// TIA Portal project "Test2" (V18)

(* hardware
DEVICE "PC-System_1"  SIMATIC PC station
   slot 0: "SIMATIC PC station"  Rail  SIMATIC PC-Station  V1.0
      slot 125: "Stationmanager"  Station_Manager  V6.0.4
   slot 1: "HMI_RT_1"  WinCC RT Professional  6AV2 105-0xxxx-xxxx  18.0.0.0
   slot 2: "IE general_1"  IE General  IE_CP  V8.2.0
      slot 1: "PROFINET interface"  IEGeneral.Interface.8.2.0
DEVICE "S7-1500/ET200MP station_1"  S7-1500 station
   slot 0: "Rail_0"  Rack  6ES7 590-1***0-0AA0
   slot 1: "PLC_2"  CPU 1511C-1 PN  6ES7 511-1CK01-0AB0  V2.9
      slot 3: "CPU display_1"  6ES7591-1AA00-0AA0
      slot 32768: "PROFINET interface_1"  X1
         slot 32769: "Port_1"  X1 P1
         slot 32770: "Port_2"  X1 P2
      slot 34817: "Virtual CP interface port_1"  Virtual CP interface port  Virtual CP interface port
*)

// ===== PLC "PLC_2"  CPU 1511C-1 PN =====

VAR_GLOBAL   // PLC tag table "Default tag table"
   "L" AT %IW2 : Int;   // уровень
   "LOV-1" AT %Q4.0 : Bool;   // КЛАПАН НА ЗАКАЧКУ ВОДЫ
   "LOV-2" AT %Q4.1 : Bool;   // Клапан на выкачку
   "tag_SpeadLminus_cm_s" AT %MD1 : Real;
   "tag_SpeadLminus_cm_s_X" AT %MD2 : Real;
   "tag_SpeadLplus_cm_s" AT %MD6 : Real;
   "tag_T1_Q" AT %M17.1 : Bool;
   "tag_T1_Start" AT %M17.0 : Bool;
END_VAR

VAR_GLOBAL   // PLC tag table "E333"
   "Auto_man_LOV-1" AT %M0.1 : Bool;   // В автоманте - 1. В ручном - 0
   "Start_stop" AT %M0.2 : Bool;   // пуск-остановка клапана закачки
   "Start_stop_2" AT %M0.3 : Bool;   // Ручное упарвеление Клапаном
   "Start_stop_Nasos" AT %M0.4 : Bool;
   "Nasos(1)" AT %M0.5 : Bool;
   "Auto_man_LOV-2" AT %M0.6 : Bool;
   "Auto_man_NASOS-1" AT %M0.7 : Bool;
   "Auto_man_ALL" AT %M10.0 : Bool;
END_VAR

DATA_BLOCK "DB_1"   // DB2
{ S7_Optimized_Access := 'FALSE' }
VERSION : 0.1
   VAR
      ResetPID : Bool;
      ManOn : Bool;
      Circle_2 : Time := T#1s;
      Circle_1 : Time := T#1s;
      Level_Sim : Real;
      SetPoin_1 : Real := 0.0;
      Gain_1 : Real := -2.0;
      Gain_2 : Real := -2.0;
      TI_1 : Time := T#20ms;
      TI_2 : Time := T#20ms;
      PID_OUT_1 : Real;
      PID_OUT_2 : Real;
      Level_Sim_Dint : DInt;
      Deadband_1 : Real;
      Deadband_2 : Real;
      PID_OUT_1_dev10 : Real;
      SpeadPLUS : Real := 1.0;
      SpeadLminus : Real := 5.0;
      PID_OUT_1_Dint : DInt;
   END_VAR
BEGIN
END_DATA_BLOCK

DATA_BLOCK "Data_E333"   // DB3
{ S7_Optimized_Access := 'TRUE' }
VERSION : 0.1
   VAR
      MAX_lvl : Real := 100.0;
      MIN_lvl : Real := 0.0;
      Pump_POWER : Real;
      MAX_Uroven : Real;
      MIN_Uroven : Real;
   END_VAR
BEGIN
END_DATA_BLOCK

DATA_BLOCK "NASOS_BD"   // DB4
{ S7_Optimized_Access := 'TRUE' }
VERSION : 0.1
   VAR
      Speed_NOW : Real;
   END_VAR
BEGIN
END_DATA_BLOCK

DATA_BLOCK "LOVs_DB"   // DB5
{ S7_Optimized_Access := 'TRUE' }
VERSION : 0.1
BEGIN
END_DATA_BLOCK

DATA_BLOCK "Avtonomiya_1"   // DB6
{ S7_Optimized_Access := 'TRUE' }
VERSION : 0.1
   VAR
      ZakachkaFlow : Real;
      OtkachkaFlow : Real;
   END_VAR
BEGIN
END_DATA_BLOCK

FUNCTION "LOV_1" : Void   // FC1, LAD
{ S7_Optimized_Access := 'TRUE' }
VERSION : 0.1
   VAR_TEMP
      "#DrainFlow_1" : Bool;
   END_VAR
BEGIN

REGION Network 1: КЛАПАН НА ЗАКАЧКУ ВОДЫ
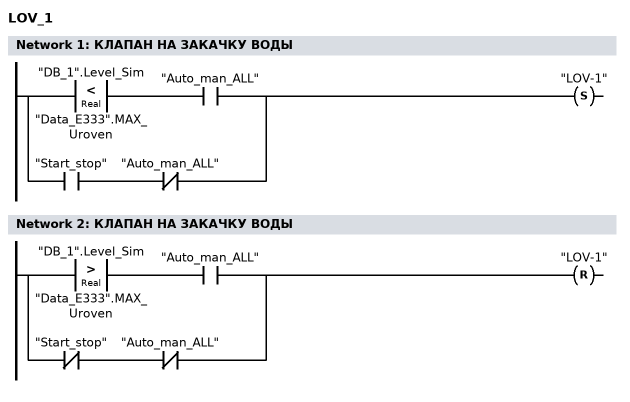
   RUNG wire#powerrail
      { S7_Templates := "SrcType := Real" } LT_Contact(in1 := "DB_1".Level_Sim, in2 := "Data_E333".MAX_Uroven)
      Contact( "Auto_man_ALL" )
      wire#w1
      S_Coil( "LOV-1" )
   END_RUNG
   RUNG wire#powerrail
      Contact( "Start_stop" )
      I_Contact( "Auto_man_ALL" )
   END_RUNG wire#w1
   // the same network as SCL:
   IF (("DB_1".Level_Sim < "Data_E333".MAX_Uroven) AND "Auto_man_ALL") OR ("Start_stop" AND NOT "Auto_man_ALL") THEN
       "LOV-1" := TRUE;
   END_IF;
END_REGION

REGION Network 2: КЛАПАН НА ЗАКАЧКУ ВОДЫ
   RUNG wire#powerrail
      { S7_Templates := "SrcType := Real" } GT_Contact(in1 := "DB_1".Level_Sim, in2 := "Data_E333".MAX_Uroven)
      Contact( "Auto_man_ALL" )
      wire#w1
      R_Coil( "LOV-1" )
   END_RUNG
   RUNG wire#powerrail
      I_Contact( "Start_stop" )
      I_Contact( "Auto_man_ALL" )
   END_RUNG wire#w1
   // the same network as SCL:
   IF (("DB_1".Level_Sim > "Data_E333".MAX_Uroven) AND "Auto_man_ALL") OR (NOT "Start_stop" AND NOT "Auto_man_ALL") THEN
       "LOV-1" := FALSE;
   END_IF;
END_REGION
END_FUNCTION

FUNCTION "FC_PID" : Void   // FC2, LAD
{ S7_Optimized_Access := 'TRUE' }
VERSION : 0.1
BEGIN

REGION Network 1
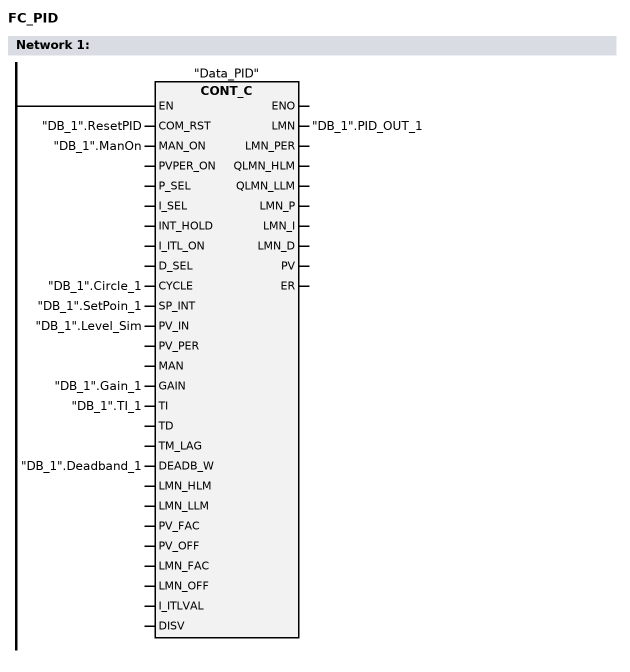
   "Data_PID"(COM_RST := "DB_1".ResetPID,   // CONT_C
              MAN_ON := "DB_1".ManOn,
              CYCLE := "DB_1".Circle_1,
              SP_INT := "DB_1".SetPoin_1,
              PV_IN := "DB_1".Level_Sim,
              GAIN := "DB_1".Gain_1,
              TI := "DB_1".TI_1,
              DEADB_W := "DB_1".Deadband_1,
              LMN => "DB_1".PID_OUT_1);
END_REGION
END_FUNCTION

FUNCTION "NASOS" : Void   // FC3, LAD
{ S7_Optimized_Access := 'TRUE' }
VERSION : 0.1
   VAR_TEMP
      PumpPower : Real;
      DrainFlow_1 : Real;
      DeltaLevel : Real;
   END_VAR
BEGIN

REGION Network 1
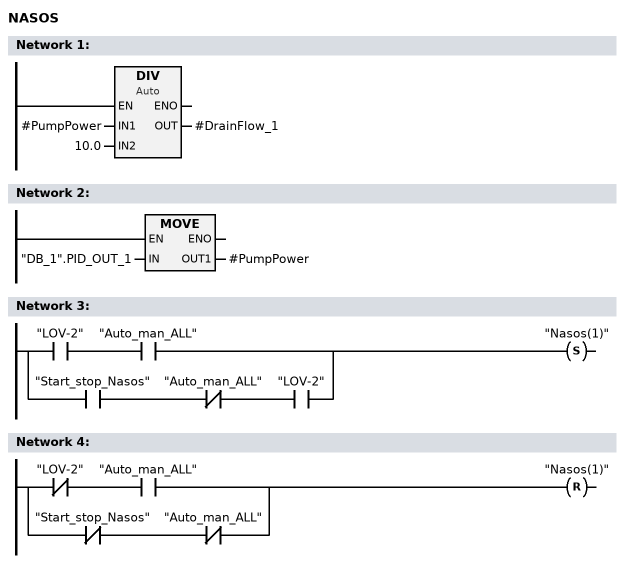
   RUNG wire#powerrail
      Div(in1 := #PumpPower, in2 := 10.0, out => #DrainFlow_1)
   END_RUNG
   // the same network as SCL:
   #DrainFlow_1 := #PumpPower / 10.0;
END_REGION

REGION Network 2
   RUNG wire#powerrail
      Move(in := "DB_1".PID_OUT_1, out1 => #PumpPower)
   END_RUNG
   // the same network as SCL:
   #PumpPower := "DB_1".PID_OUT_1;
END_REGION

REGION Network 3
   RUNG wire#powerrail
      Contact( "LOV-2" )
      Contact( "Auto_man_ALL" )
      wire#w1
      S_Coil( "Nasos(1)" )
   END_RUNG
   RUNG wire#powerrail
      Contact( "Start_stop_Nasos" )
      I_Contact( "Auto_man_ALL" )
      Contact( "LOV-2" )
   END_RUNG wire#w1
   // the same network as SCL:
   IF ("LOV-2" AND "Auto_man_ALL") OR ("Start_stop_Nasos" AND NOT "Auto_man_ALL" AND "LOV-2") THEN
       "Nasos(1)" := TRUE;
   END_IF;
END_REGION

REGION Network 4
   RUNG wire#powerrail
      I_Contact( "LOV-2" )
      Contact( "Auto_man_ALL" )
      wire#w1
      R_Coil( "Nasos(1)" )
   END_RUNG
   RUNG wire#powerrail
      I_Contact( "Start_stop_Nasos" )
      I_Contact( "Auto_man_ALL" )
   END_RUNG wire#w1
   // the same network as SCL:
   IF (NOT "LOV-2" AND "Auto_man_ALL") OR (NOT "Start_stop_Nasos" AND NOT "Auto_man_ALL") THEN
       "Nasos(1)" := FALSE;
   END_IF;
END_REGION

REGION Network 5 (SCL)
   "DB_1".Level_Sim := "DB_1".Level_Sim + ("Avtonomiya_1".ZakachkaFlow / 60.0) * 0.1
   - ("Avtonomiya_1".OtkachkaFlow  / 60.0) * ("DB_1".PID_OUT_1 / 100.0) * 0.1;

   "NASOS_BD".Speed_NOW := "Avtonomiya_1".OtkachkaFlow * ("DB_1".PID_OUT_1 / 100.0);


   "Data_E333".Pump_POWER := #PumpPower;
END_REGION
END_FUNCTION

FUNCTION "LOV_2" : Void   // FC4, LAD
{ S7_Optimized_Access := 'TRUE' }
VERSION : 0.1
BEGIN

REGION Network 1: Клапан на выкачку
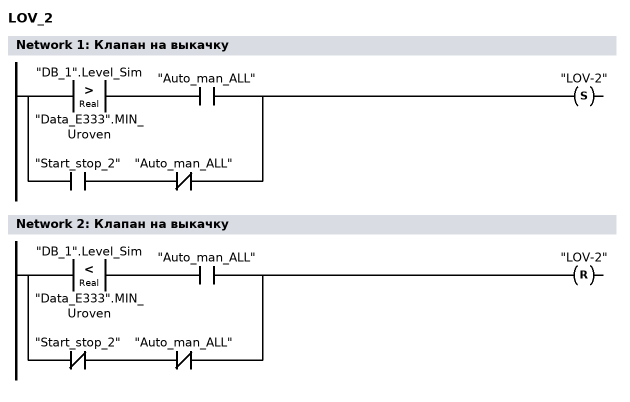
   RUNG wire#powerrail
      { S7_Templates := "SrcType := Real" } GT_Contact(in1 := "DB_1".Level_Sim, in2 := "Data_E333".MIN_Uroven)
      Contact( "Auto_man_ALL" )
      wire#w1
      S_Coil( "LOV-2" )
   END_RUNG
   RUNG wire#powerrail
      Contact( "Start_stop_2" )
      I_Contact( "Auto_man_ALL" )
   END_RUNG wire#w1
   // the same network as SCL:
   IF (("DB_1".Level_Sim > "Data_E333".MIN_Uroven) AND "Auto_man_ALL") OR ("Start_stop_2" AND NOT "Auto_man_ALL") THEN
       "LOV-2" := TRUE;
   END_IF;
END_REGION

REGION Network 2: Клапан на выкачку
   RUNG wire#powerrail
      { S7_Templates := "SrcType := Real" } LT_Contact(in1 := "DB_1".Level_Sim, in2 := "Data_E333".MIN_Uroven)
      Contact( "Auto_man_ALL" )
      wire#w1
      R_Coil( "LOV-2" )
   END_RUNG
   RUNG wire#powerrail
      I_Contact( "Start_stop_2" )
      I_Contact( "Auto_man_ALL" )
   END_RUNG wire#w1
   // the same network as SCL:
   IF (("DB_1".Level_Sim < "Data_E333".MIN_Uroven) AND "Auto_man_ALL") OR (NOT "Start_stop_2" AND NOT "Auto_man_ALL") THEN
       "LOV-2" := FALSE;
   END_IF;
END_REGION
END_FUNCTION

FUNCTION "Avtonomiya" : Void   // FC5, LAD
{ S7_Optimized_Access := 'TRUE' }
VERSION : 0.1
BEGIN

REGION Network 1
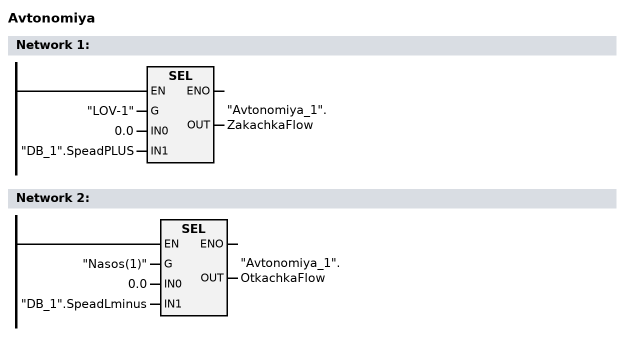
   "Avtonomiya_1".ZakachkaFlow := SEL(G := "LOV-1", IN0 := 0.0, IN1 := "DB_1".SpeadPLUS);
END_REGION

REGION Network 2
   "Avtonomiya_1".OtkachkaFlow := SEL(G := "Nasos(1)", IN0 := 0.0, IN1 := "DB_1".SpeadLminus);
END_REGION
END_FUNCTION

ORGANIZATION_BLOCK "Main"   // OB1, LAD, ProgramCycle
TITLE = "Main Program Sweep (Cycle)"
{ S7_Optimized_Access := 'TRUE' }
VERSION : 0.1
   VAR_INPUT
      Initial_Call : Bool;   // Initial call of this OB
      Remanence : Bool;   // =True, if remanent data are available
   END_VAR
   VAR_TEMP
      Temp : Real;
   END_VAR
BEGIN
END_ORGANIZATION_BLOCK

ORGANIZATION_BLOCK "PID_1"   // OB123, LAD, ProgramCycle
TITLE = "Main Program Sweep (Cycle)"
{ S7_Optimized_Access := 'TRUE' }
VERSION : 0.1
   VAR_INPUT
      Initial_Call : Bool;   // Initial call of this OB
      Remanence : Bool;   // =True, if remanent data are available
   END_VAR
BEGIN

REGION Network 1
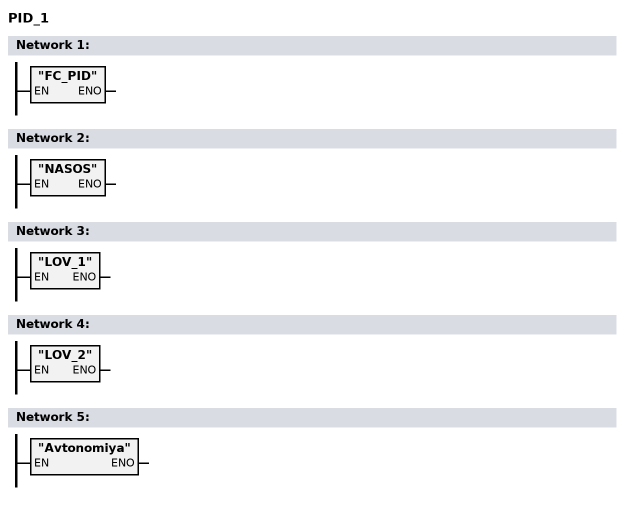
   RUNG wire#powerrail
      "FC_PID"()
   END_RUNG
   // the same network as SCL:
   "FC_PID"();
END_REGION

REGION Network 2
   RUNG wire#powerrail
      "NASOS"()
   END_RUNG
   // the same network as SCL:
   "NASOS"();
END_REGION

REGION Network 3
   RUNG wire#powerrail
      "LOV_1"()
   END_RUNG
   // the same network as SCL:
   "LOV_1"();
END_REGION

REGION Network 4
   RUNG wire#powerrail
      "LOV_2"()
   END_RUNG
   // the same network as SCL:
   "LOV_2"();
END_REGION

REGION Network 5
   RUNG wire#powerrail
      "Avtonomiya"()
   END_RUNG
   // the same network as SCL:
   "Avtonomiya"();
END_REGION
END_ORGANIZATION_BLOCK

(* ===== HMI "HMI_RT_1" =====
system functions are stored by id; their names below are inferred from use
connection "HMI_Connection_2": S71200_TCP_IP, SCADA_S7_1500_OMS
connection "HMI_Connection_3": S71200_TCP_IP, SCADA_S7_1500_OMS

HMI tags "Default tag table"
   "LOV-1" : Bool = PLC "LOV-1" AT %Q4.0, 500 ms
   "Auto_man_LOV-1_HMI" : Bool = PLC "Auto_man_LOV-1" AT %M0.1, 500 ms
   "Start_stop_LOV-1_HMI" : Bool = PLC Start_stop AT %M0.2, 500 ms
   "LOV-2" : Bool = PLC "LOV-2" AT %Q4.1, 500 ms
   "Start_stop_LOV-2_HMI" : Bool = PLC Start_stop_2 AT %M0.3, 500 ms
   "Auto_Nasos" : Bool = PLC "Nasos(1)" AT %M0.5, 500 ms
   "ResetPID" : Bool = PLC DB_1.ResetPID AT %DB2.DBX0.0, 500 ms
   "ManOn" : Bool = PLC DB_1.ManOn AT %DB2.DBX0.1, 500 ms
   "Circle_1" : Time = PLC DB_1.Circle_1 AT %DB2.DBD6, 500 ms
   "Circle_2" : Time = PLC DB_1.Circle_2 AT %DB2.DBD2, 500 ms
   "Level_Sim" : Real = PLC DB_1.Level_Sim AT %DB2.DBD10, 500 ms
   "SetPoin_1" : Real = PLC DB_1.SetPoin_1 AT %DB2.DBD14, 500 ms
   "Gain_1" : Real = PLC DB_1.Gain_1 AT %DB2.DBD18, 500 ms
   "Gain_2" : Real = PLC DB_1.Gain_2 AT %DB2.DBD22, 500 ms
   "TI_1_HMI" : Time = PLC DB_1.TI_1 AT %DB2.DBD26, 500 ms
   "TI_2_HMI" : Time = PLC DB_1.TI_2 AT %DB2.DBD30, 500 ms
   "PID_OUT_1" : Real = PLC DB_1.PID_OUT_1 AT %DB2.DBD34, 500 ms
   "PID_OUT_2" : Real = PLC DB_1.PID_OUT_2 AT %DB2.DBD38, 500 ms
   "Level_Sim_Dint" : DInt = PLC DB_1.Level_Sim_Dint AT %DB2.DBD42, 500 ms
   "Deadband_1" : Real = PLC DB_1.Deadband_1 AT %DB2.DBD46, 500 ms
   "Deadband_2" : Real = PLC DB_1.Deadband_2 AT %DB2.DBD50, 500 ms
   "PID_OUT_1_dev10" : Real = PLC DB_1.PID_OUT_1_dev10 AT %DB2.DBD54, 500 ms
   "SpeadPLUS" : Real = PLC Avtonomiya_1.ZakachkaFlow AT %DB2.DBD58, 500 ms
   "SpeadLminus" : Real = PLC DB_1.SpeadLminus AT %DB2.DBD62, 500 ms
   "PID_OUT_1_Dint" : DInt = PLC DB_1.PID_OUT_1_Dint AT %DB2.DBD66, 500 ms
   "Data_E333_MAX_lvl" : Real = PLC Data_E333.MAX_lvl, 500 ms
   "Data_E333_MIN_lvl" : Real = PLC Data_E333.MIN_lvl, 500 ms
   "Pump_POWER" : Real = PLC Data_E333.Pump_POWER AT %DB1.DBD0, 500 ms
   "NASOS_BD_Speed_NOW" : Real = PLC NASOS_BD.Speed_NOW, 500 ms
   "Auto_man_NASOS-1" : Bool = PLC "Auto_man_NASOS-1" AT %M0.7, 500 ms

HMI tags "E333"
   "MAX_Uroven" : Real = PLC Data_E333.MAX_Uroven AT %DB1.DBW0, 500 ms
   "MIN_Uroven" : Real = PLC Data_E333.MIN_Uroven, 500 ms
   "Auto_man_ALL" : Bool = PLC Auto_man_ALL AT %M10.0, 500 ms

HMI tags "NASOS"
   "NASOS_HMI" : Bool = PLC "Nasos(1)" AT %M0.5, 500 ms
   "Auto_man_NASOS-1_HMI" : Bool = PLC "Auto_man_NASOS-1" AT %M0.7, 500 ms
   "Start_stop_Nasos_HMI" : Bool = PLC Start_stop_Nasos AT %M0.4, 500 ms
   "Auto_man_LOV-2_HMI" : Bool = PLC "Auto_man_LOV-2" AT %M0.6, 500 ms

screen "Screen_1" 2000x800
   TextField "Text field_5" at 199,311 size 42x14; Text 'LOV - 2'
   Group "Group_5" at 201,328 size 30x33
   TextField "Text field_4" at 270,310 size 108x14; Text '50WQH-10-10-0.75'
   Group "Group_8" at 296,329 size 48x48
      on Click: function_c00bc162("Screen_1", "Screen window_3", Visible, '1')
   Group "Group_7" at 296,329 size 48x48
      on Click: function_c00bc162("Screen_1", "Screen window_3", Visible, '1')
      Visibility <- "NASOS_HMI"
   ScreenWindow "Screen window_3" at 0,425 size 616x280; CaptionText '50WQH-10-10-0.75'; ScreenName "PupUP_AI-1"
   OnlineTrendControl "f(t) trend view_1" at 621,470 size 640x335
   Group "Group_3" at 72,46 size 30x33
      on Click: function_c00bc162("Screen_1", "Screen window_1", Visible, '1')
   Group "Group_10" at 199,328 size 33x33
      Visibility <- "LOV-2"
   Group "Group_6" at 71,46 size 32x33
      Visibility <- "LOV-1"
      on Click: function_c00bc162("Screen_1", "Screen window_1", Visible, '1')
   TextField "Text field_1" at 69,28 size 42x14; Text 'LOV - 1'
   ScreenWindow "Screen window_2" at 406,179 size 227x181; ScreenName "E333"
   Group "Group" at 127,125 size 62x163
      on Click: function_c00bc162("Screen_1", "Screen window_2", Visible, '1')
   ScreenWindow "Screen window_1" at 0,97 size 165x97; ScreenName "PupUp_LOV-1"; CaptionText 'LOV - 1'
   ScreenWindow "Screen window_4" at 0,302 size 164x97; ScreenName "PupUp_LOV-2"; CaptionText 'PupUp_LOV-2'
   TextField "Text field_2" at 308,142 size 24x14; Text 'ПИД'
   TextField "Text field_6" at 287,157 size 68x14; Text 'LICA 103-01'
   Group "Group_11" at 273,175 size 19x19
      on Click: ResetBit("Auto_man_ALL")
   Group "Group_12" at 273,175 size 19x19
      on Click: SetBit("Auto_man_ALL")
      Visibility <- "Auto_man_ALL"
   Rectangle "Rectangle_1" at 127,156 size 62x132
      on Click: function_c00bc162("Screen_1", "Screen window_3", Visible, '1')
   CircleSegment "Circle segment_1" at 127,125 size 62x31
   TextField "Text field_3" at 138,190 size 42x21; Text 'E 333'
   CircleSegment "Circle segment_3" at 81,46 size 14x7
   Group "Group_2" at 71,59 size 32x20
   CircleSegment "Circle segment_4" at 210,328 size 14x7
   Group "Group_4" at 201,341 size 30x20
   CircleSegment "Circle segment_2" at 81,46 size 14x7
   Group "Group_1" at 72,59 size 30x20
   CircleSegment "Circle segment_5" at 209,328 size 14x7
   Group "Group_9" at 199,341 size 33x20
   HmiScreenItemData "Button_1" at 0,0 size 0x0
   HmiScreenItemData "Button_6" at 0,0 size 0x0
   TextField "Text field_7" at 278,177 size 10x14; Text 'A'
   TextField "Text field_8" at 278,177 size 10x14; Text 'M'

screen "PupUp_LOV-1" 155x170
   Button "Button_4" at 4,55 size 69x24; TextOff 'ОТКРЫТЬ'
      on Click: SetBit("Start_stop_LOV-1_HMI")
   Button "Button_5" at 82,56 size 69x24; TextOff 'ЗАКРЫТЬ'
      on Click: ResetBit("Start_stop_LOV-1_HMI")
   Button "Button_1" at 125,1 size 28x25; TextOff 'X'
      on Click: function_c00bc162("Screen_1", "Screen window_1", Visible, '0')
   TextField "Text field_1" at 6,4 size 51x22; Text 'LOV-1'
   TextField "Text field_2" at 19,32 size 115x18; Text 'РУЧНОЙ РЕЖИМ'

screen "PupUp_LOV-2" 155x170
   Button "Button_4" at 5,55 size 69x24; TextOff 'ОТКРЫТЬ'
      on Click: SetBit("Start_stop_LOV-2_HMI")
   Button "Button_5" at 80,55 size 69x24; TextOff 'ЗАКРЫТЬ'
      on Click: ResetBit("Start_stop_LOV-2_HMI")
   Button "Button_1" at 125,0 size 28x25; TextOff 'X'
      on Click: function_c00bc162("Screen_1", "Screen window_1", Visible, '0')
   TextField "Text field_1" at 6,3 size 51x22; Text 'LOV-2'
   TextField "Text field_2" at 19,32 size 115x18; Text 'РУЧНОЙ РЕЖИМ'

screen "PupUP_AI-1" 800x600
   Button "Button_5" at 577,1 size 28x25; TextOff 'X'
      on Click: function_c00bc162("Screen_1", "Screen window_3", Visible, '0')
   TextField "Text field_10" at 6,4 size 151x22; Text '50WQH-10-10-0.75'
   Button "Button_3" at 21,193 size 55x23; TextOff 'Старт'
      on Click: SetBit("Start_stop_Nasos_HMI")
   Button "Button_4" at 102,194 size 55x22; TextOff 'Стоп'
      on Click: ResetBit("Start_stop_Nasos_HMI")
   IOField "I/O field_1" at 314,31 size 80x20; FormatPattern 999
      ProcessValue <- "SetPoin_1"
   TextField "Text field_2" at 412,31 size 145x18; Text 'Уставка (SetPoint)'
   IOField "I/O field_2" at 314,59 size 80x20; FormatPattern 999
      ProcessValue <- "SpeadPLUS"
   TextField "Text field_3" at 411,58 size 177x18; Text 'Скорость ПОПОЛНЕИЯ'
   IOField "I/O field_3" at 314,89 size 80x20; FormatPattern 999
      ProcessValue <- "SpeadLminus"
   TextField "Text field_4" at 411,89 size 130x18; Text 'Скорость СЛИВА'
   TextField "Text field_5" at 372,31 size 19x18; Text 'см'
   TextField "Text field_6" at 345,61 size 46x14; Text 'см/мин'
   Gauge "Gauge_1" at 186,166 size 106x106; CaptionText '%'
      MaximumValue <- "Data_E333_MAX_lvl"
      MinimumValue <- "Data_E333_MIN_lvl"
      ProcessValue <- "Pump_POWER"
   TextField "Text field_8" at 183,154 size 119x14; Text 'мощность насоса'
   TextField "Text field_7" at 345,91 size 46x14; Text 'см/мин'
   TextField "Text field_16" at 367,188 size 171x17; Text 'Емкость заполненно %'
   TextField "Text field_21" at 361,171 size 177x17; Text 'Скорость слива см/мин'
   TextField "Text field_1" at 314,154 size 224x17; Text 'Скорость пополнения см/мин'
   IOField "I/O field_4" at 11,30 size 80x20; FormatPattern 999
      ProcessValue <- "Gain_1"
   IOField "I/O field_5" at 10,60 size 80x20; FormatPattern 999
      ProcessValue <- "TI_1_HMI"
   IOField "I/O field_6" at 10,89 size 80x20; FormatPattern 999
      ProcessValue <- "Circle_1"
   IOField "I/O field_7" at 10,117 size 80x20; FormatPattern 999
      ProcessValue <- "Deadband_1"
   TextField "Text field_9" at 110,32 size 69x18; Text 'П (GAIN)'
   TextField "Text field_11" at 110,62 size 63x18; Text 'И (TI), s'
   TextField "Text field_13" at 114,89 size 10x18; Text 'Text'
   TextField "Text field_15" at 110,89 size 124x18; Text 'Цикл (CYKLE),s'
   TextField "Text field_17" at 110,116 size 190x18; Text 'Мертвая зона (DEAD_W)'
   IOField "I/O field_9" at 550,155 size 53x20; FormatPattern s999999999.999
      ProcessValue <- "SpeadPLUS"
   IOField "I/O field_10" at 550,173 size 54x20; FormatPattern s999999999.999
      ProcessValue <- "NASOS_BD_Speed_NOW"
   IOField "I/O field_11" at 550,189 size 55x20; FormatPattern s999999999.999
      ProcessValue <- "Level_Sim"
   Button "Button_6" at 369,221 size 194x30; TextOff 'Отобразить график'
      on Click: function_c00bc162("Screen_1", "f(t) trend view_1", Visible, '1')
   TextField "Text field_12" at 37,158 size 115x18; Text 'РУЧНОЙ РЕЖИМ'
   TextField "Text field_18" at 23,224 size 156x32; Text 'LOV-2 ЗАКРЫТ НАСОС НЕ ЗАПУСТИТСЯ'
      Visibility <- "LOV-2"

screen "E333" 250x190
   Button "Button_1" at 187,2 size 28x25; TextOff 'X'
      on Click: function_c00bc162("Screen_1", "Screen window_2", Visible, '0')
   Bar "Bar_1" at 1,27 size 105x143; MinimumValue 0; MaximumValue 100
      MinimumValue <- "Data_E333_MIN_lvl"
      ProcessValue <- "Level_Sim"
      MaximumValue <- "Data_E333_MAX_lvl"
   TextField "Text field_1" at 6,4 size 37x22; Text 'E333'
   IOField "I/O field_1" at 109,60 size 107x20; FormatPattern 999
      ProcessValue <- "MAX_Uroven"
   TextField "Text field_2" at 110,34 size 106x18; Text 'MAX. Уровень'
   TextField "Text field_3" at 111,110 size 105x18; Text 'MIN. Уровень'
   IOField "I/O field_2" at 111,133 size 107x20; FormatPattern 999
      ProcessValue <- "MIN_Uroven"
*)

(* ===== HMI "HMI_RT_1" =====

ScreenModuleEditorView "Faceplate_1_S2tandard_Pump" 1024x768
   Group "Group" at 0,0 size 40x25
*)